// TIA Portal V17 export
// export: Created 2025-03-10T13:09:50.3447093Z, ExportSetting WithDefaults, DisplayName Totally Integrated Automation Portal, DisplayVersion V17 Update 8, DisplayName TIA Portal Openness, DisplayVersion V17 Update 8, DisplayName TIA Portal Version Control Interface, DisplayVersion V17, DisplayName SINAMICS Startdrive Advanced, DisplayVersion V17 SP2, DisplayName SINAMICS Startdrive G110M, G120, G120C, G120D, G120P, G115D, DisplayVersion V17 SP2, DisplayName SINAMICS Startdrive G130, G150, S120, S150, SINAMICS MV, S210, DisplayVersion V17 SP2, DisplayName STEP 7 Professional, DisplayVersion V17 Update 8, DisplayName SINUMERIK ONE STEP 7 Toolbox, DisplayVersion V17 Update 12, DisplayName SINUMERIK 840D sl STEP 7 Toolbox, DisplayVersion V17 Update 12, DisplayName STEP 7 Safety, DisplayVersion V17 Update 6, DisplayName WinCC Advanced, DisplayVersion V17 Update 8
FUNCTION "FC8004_UNIT_03_CLADDING" : Void   // FC8004, LAD
{ S7_Optimized_Access := 'FALSE' }
AUTHOR : ETXETAR
VERSION : 1.0
// stored: AutoNumber false, IsIECCheckEnabled false, SetENOAutomatically false, UDAEnableTagReadback false
   VAR_TEMP
      ZERO : Byte;   // ZERO
      STATUS_BLKMOV : Int;   // STATUS BLKMOV
      STATUS_FILL : Int;   // STATUS FILL
   END_VAR
   VAR CONSTANT
      FC_NUMBER : DInt := 8004;   // FC NUMBER
   END_VAR
   VAR_TEMP   // added for the SCL form of the ladder/FBD networks
      _w1 : Bool;
      _w2 : Bool;
      _w3 : Bool;
      _w4 : Bool;
   END_VAR
BEGIN

REGION Network 1: ZERO
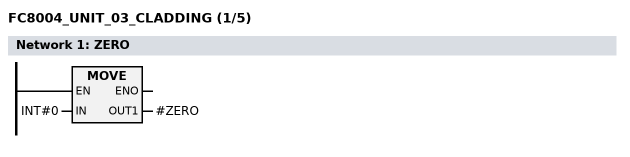
   RUNG wire#powerrail
      { S7_GenerateENO := "TRUE" } Move(in := INT#0, out1 => #ZERO)
   END_RUNG
   // the same network as SCL:
   #ZERO := INT#0;
END_REGION

REGION Network 2: HMI MANUAL PART A FIXTURE 1 STATUS
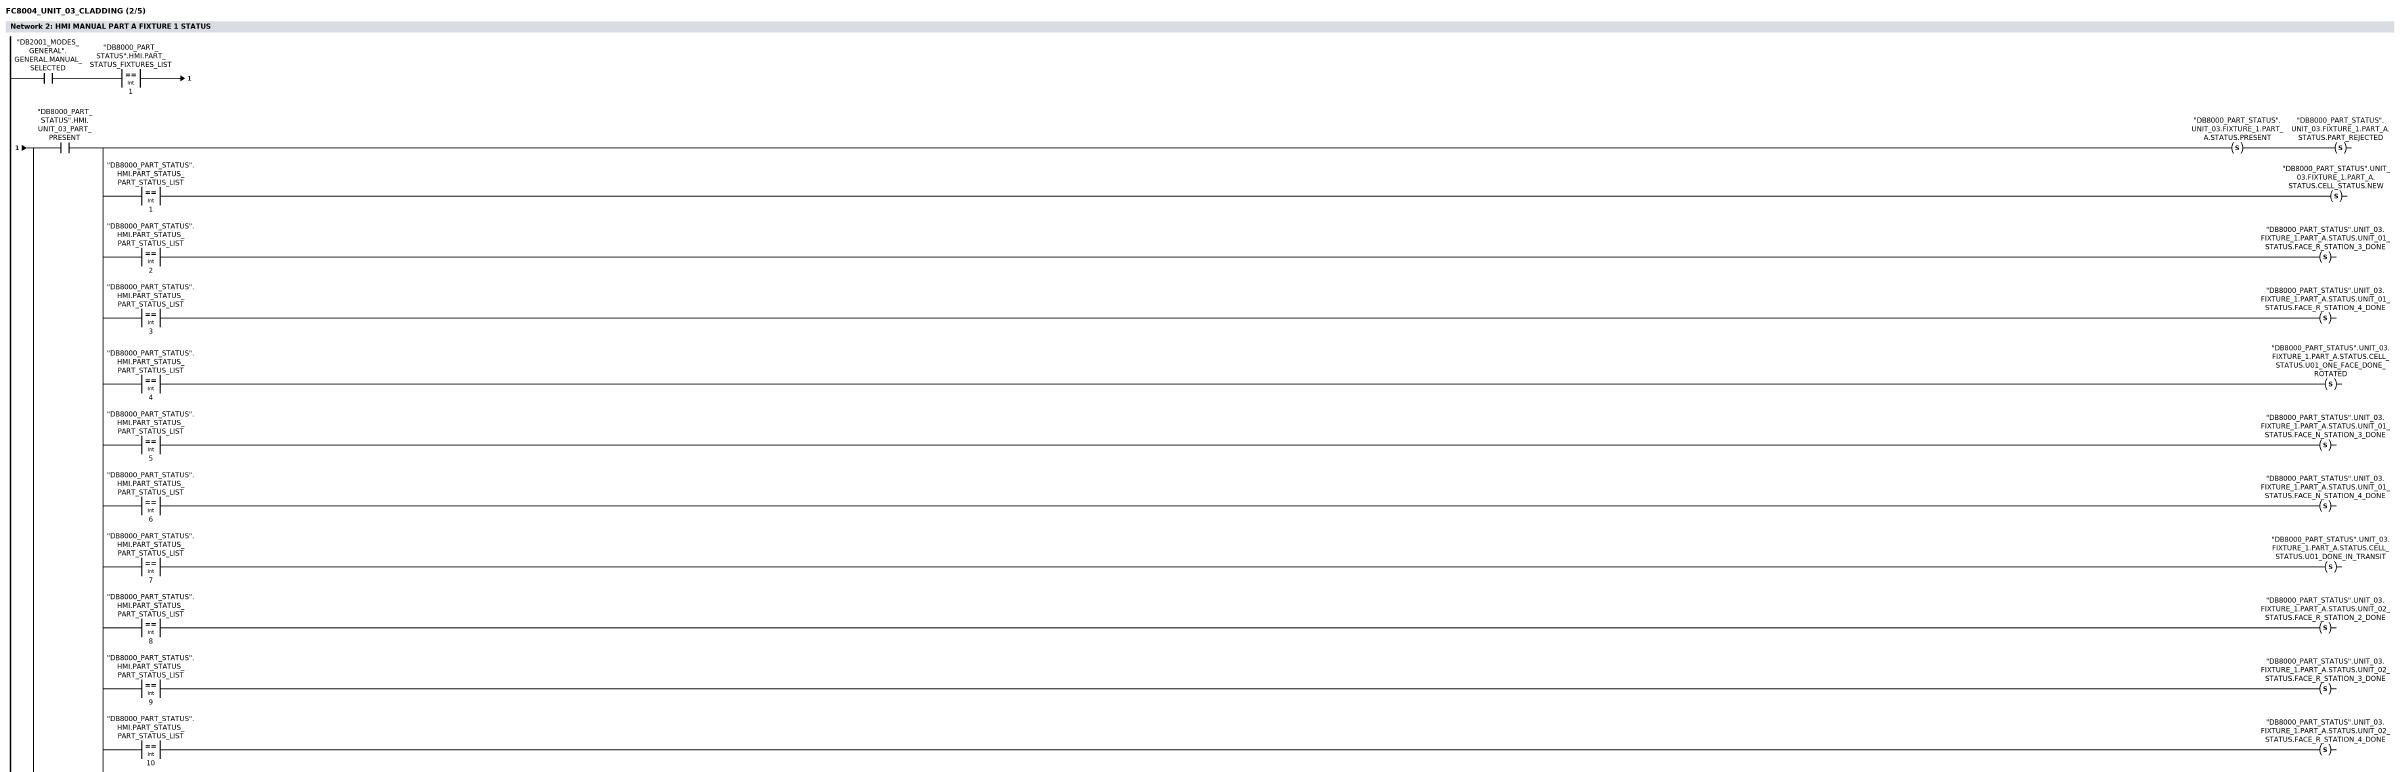
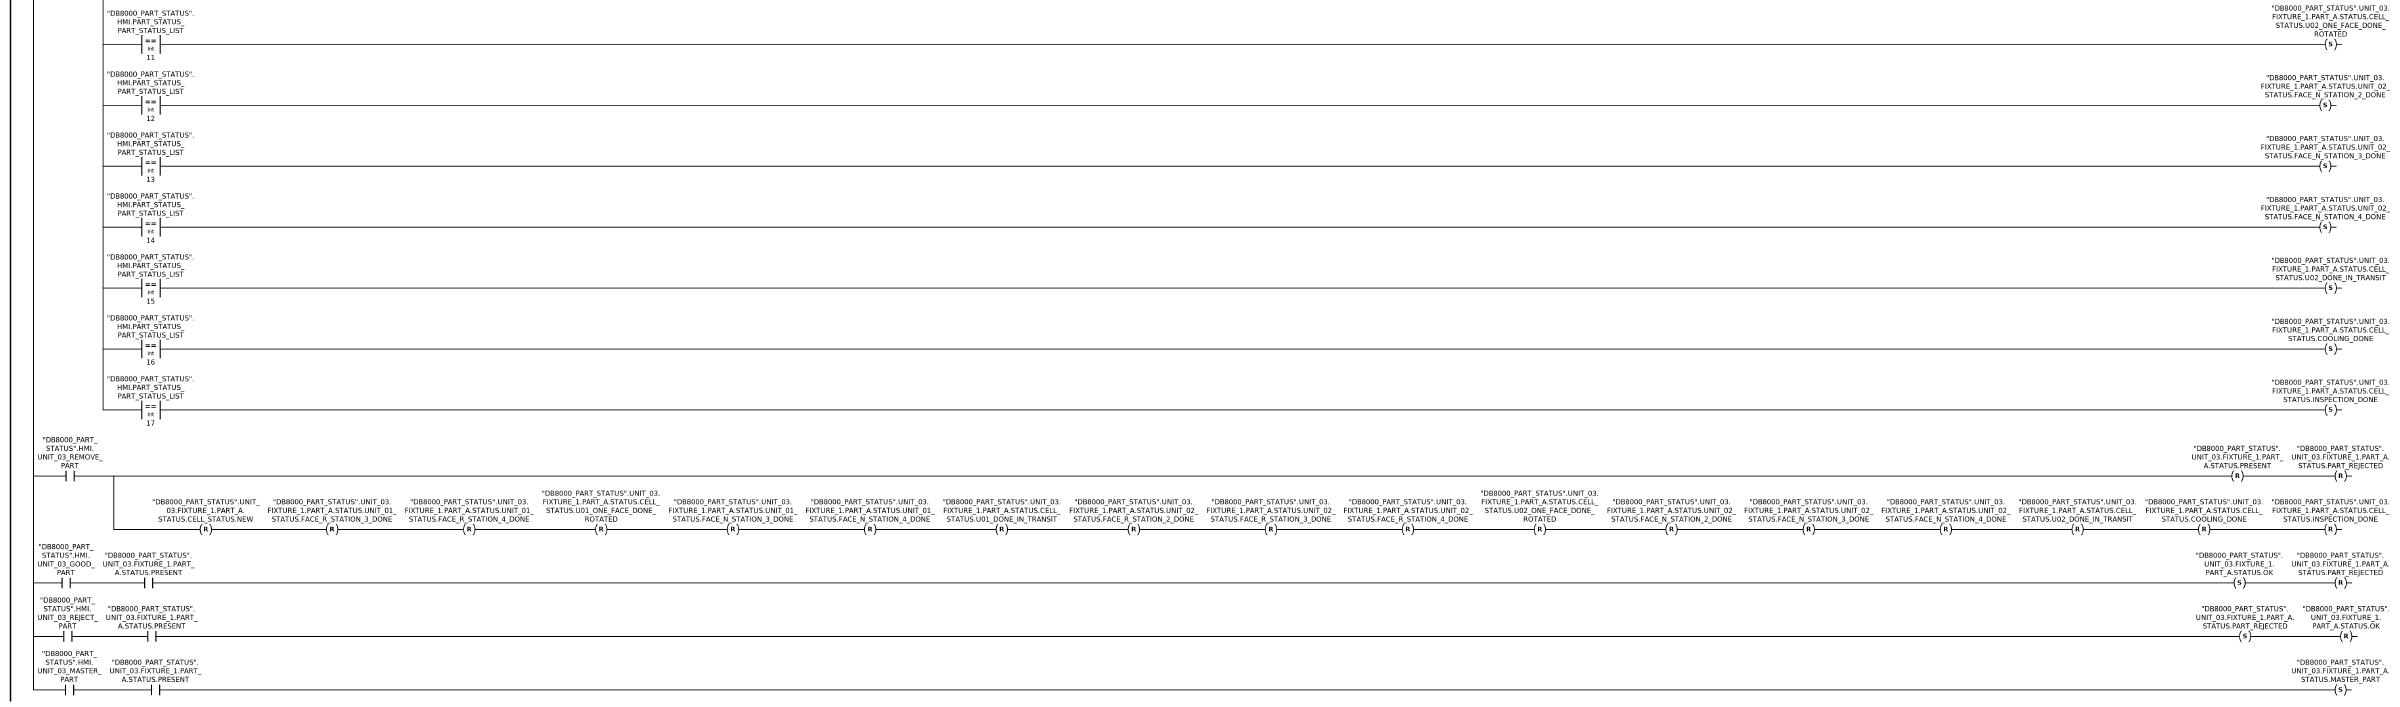
   RUNG wire#powerrail
      Contact( "DB2001_MODES_GENERAL".GENERAL.MANUAL_SELECTED )
      { S7_Templates := "SrcType := Int" } EQ_Contact(in1 := "DB8000_PART_STATUS".HMI.PART_STATUS_FIXTURES_LIST, in2 := 1)
      wire#w1
      Contact( "DB8000_PART_STATUS".HMI.UNIT_03_PART_PRESENT )
      wire#w2
      S_Coil( "DB8000_PART_STATUS".UNIT_03.FIXTURE_1.PART_A.STATUS.PRESENT )
      S_Coil( "DB8000_PART_STATUS".UNIT_03.FIXTURE_1.PART_A.STATUS.PART_REJECTED )
   END_RUNG
   RUNG wire#w2
      { S7_Templates := "SrcType := Int" } EQ_Contact(in1 := "DB8000_PART_STATUS".HMI.PART_STATUS_PART_STATUS_LIST, in2 := 1)
      S_Coil( "DB8000_PART_STATUS".UNIT_03.FIXTURE_1.PART_A.STATUS.CELL_STATUS.NEW )
   END_RUNG
   RUNG wire#w2
      { S7_Templates := "SrcType := Int" } EQ_Contact(in1 := "DB8000_PART_STATUS".HMI.PART_STATUS_PART_STATUS_LIST, in2 := 2)
      S_Coil( "DB8000_PART_STATUS".UNIT_03.FIXTURE_1.PART_A.STATUS.UNIT_01_STATUS.FACE_R_STATION_3_DONE )
   END_RUNG
   RUNG wire#w2
      { S7_Templates := "SrcType := Int" } EQ_Contact(in1 := "DB8000_PART_STATUS".HMI.PART_STATUS_PART_STATUS_LIST, in2 := 3)
      S_Coil( "DB8000_PART_STATUS".UNIT_03.FIXTURE_1.PART_A.STATUS.UNIT_01_STATUS.FACE_R_STATION_4_DONE )
   END_RUNG
   RUNG wire#w2
      { S7_Templates := "SrcType := Int" } EQ_Contact(in1 := "DB8000_PART_STATUS".HMI.PART_STATUS_PART_STATUS_LIST, in2 := 4)
      S_Coil( "DB8000_PART_STATUS".UNIT_03.FIXTURE_1.PART_A.STATUS.CELL_STATUS.U01_ONE_FACE_DONE_ROTATED )
   END_RUNG
   RUNG wire#w2
      { S7_Templates := "SrcType := Int" } EQ_Contact(in1 := "DB8000_PART_STATUS".HMI.PART_STATUS_PART_STATUS_LIST, in2 := 5)
      S_Coil( "DB8000_PART_STATUS".UNIT_03.FIXTURE_1.PART_A.STATUS.UNIT_01_STATUS.FACE_N_STATION_3_DONE )
   END_RUNG
   RUNG wire#w2
      { S7_Templates := "SrcType := Int" } EQ_Contact(in1 := "DB8000_PART_STATUS".HMI.PART_STATUS_PART_STATUS_LIST, in2 := 6)
      S_Coil( "DB8000_PART_STATUS".UNIT_03.FIXTURE_1.PART_A.STATUS.UNIT_01_STATUS.FACE_N_STATION_4_DONE )
   END_RUNG
   RUNG wire#w2
      { S7_Templates := "SrcType := Int" } EQ_Contact(in1 := "DB8000_PART_STATUS".HMI.PART_STATUS_PART_STATUS_LIST, in2 := 7)
      S_Coil( "DB8000_PART_STATUS".UNIT_03.FIXTURE_1.PART_A.STATUS.CELL_STATUS.U01_DONE_IN_TRANSIT )
   END_RUNG
   RUNG wire#w2
      { S7_Templates := "SrcType := Int" } EQ_Contact(in1 := "DB8000_PART_STATUS".HMI.PART_STATUS_PART_STATUS_LIST, in2 := 8)
      S_Coil( "DB8000_PART_STATUS".UNIT_03.FIXTURE_1.PART_A.STATUS.UNIT_02_STATUS.FACE_R_STATION_2_DONE )
   END_RUNG
   RUNG wire#w2
      { S7_Templates := "SrcType := Int" } EQ_Contact(in1 := "DB8000_PART_STATUS".HMI.PART_STATUS_PART_STATUS_LIST, in2 := 9)
      S_Coil( "DB8000_PART_STATUS".UNIT_03.FIXTURE_1.PART_A.STATUS.UNIT_02_STATUS.FACE_R_STATION_3_DONE )
   END_RUNG
   RUNG wire#w2
      { S7_Templates := "SrcType := Int" } EQ_Contact(in1 := "DB8000_PART_STATUS".HMI.PART_STATUS_PART_STATUS_LIST, in2 := 10)
      S_Coil( "DB8000_PART_STATUS".UNIT_03.FIXTURE_1.PART_A.STATUS.UNIT_02_STATUS.FACE_R_STATION_4_DONE )
   END_RUNG
   RUNG wire#w2
      { S7_Templates := "SrcType := Int" } EQ_Contact(in1 := "DB8000_PART_STATUS".HMI.PART_STATUS_PART_STATUS_LIST, in2 := 11)
      S_Coil( "DB8000_PART_STATUS".UNIT_03.FIXTURE_1.PART_A.STATUS.CELL_STATUS.U02_ONE_FACE_DONE_ROTATED )
   END_RUNG
   RUNG wire#w2
      { S7_Templates := "SrcType := Int" } EQ_Contact(in1 := "DB8000_PART_STATUS".HMI.PART_STATUS_PART_STATUS_LIST, in2 := 12)
      S_Coil( "DB8000_PART_STATUS".UNIT_03.FIXTURE_1.PART_A.STATUS.UNIT_02_STATUS.FACE_N_STATION_2_DONE )
   END_RUNG
   RUNG wire#w2
      { S7_Templates := "SrcType := Int" } EQ_Contact(in1 := "DB8000_PART_STATUS".HMI.PART_STATUS_PART_STATUS_LIST, in2 := 13)
      S_Coil( "DB8000_PART_STATUS".UNIT_03.FIXTURE_1.PART_A.STATUS.UNIT_02_STATUS.FACE_N_STATION_3_DONE )
   END_RUNG
   RUNG wire#w2
      { S7_Templates := "SrcType := Int" } EQ_Contact(in1 := "DB8000_PART_STATUS".HMI.PART_STATUS_PART_STATUS_LIST, in2 := 14)
      S_Coil( "DB8000_PART_STATUS".UNIT_03.FIXTURE_1.PART_A.STATUS.UNIT_02_STATUS.FACE_N_STATION_4_DONE )
   END_RUNG
   RUNG wire#w2
      { S7_Templates := "SrcType := Int" } EQ_Contact(in1 := "DB8000_PART_STATUS".HMI.PART_STATUS_PART_STATUS_LIST, in2 := 15)
      S_Coil( "DB8000_PART_STATUS".UNIT_03.FIXTURE_1.PART_A.STATUS.CELL_STATUS.U02_DONE_IN_TRANSIT )
   END_RUNG
   RUNG wire#w2
      { S7_Templates := "SrcType := Int" } EQ_Contact(in1 := "DB8000_PART_STATUS".HMI.PART_STATUS_PART_STATUS_LIST, in2 := 16)
      S_Coil( "DB8000_PART_STATUS".UNIT_03.FIXTURE_1.PART_A.STATUS.CELL_STATUS.COOLING_DONE )
   END_RUNG
   RUNG wire#w2
      { S7_Templates := "SrcType := Int" } EQ_Contact(in1 := "DB8000_PART_STATUS".HMI.PART_STATUS_PART_STATUS_LIST, in2 := 17)
      S_Coil( "DB8000_PART_STATUS".UNIT_03.FIXTURE_1.PART_A.STATUS.CELL_STATUS.INSPECTION_DONE )
   END_RUNG
   RUNG wire#w1
      Contact( "DB8000_PART_STATUS".HMI.UNIT_03_REMOVE_PART )
      wire#w3
      R_Coil( "DB8000_PART_STATUS".UNIT_03.FIXTURE_1.PART_A.STATUS.PRESENT )
      R_Coil( "DB8000_PART_STATUS".UNIT_03.FIXTURE_1.PART_A.STATUS.PART_REJECTED )
   END_RUNG
   RUNG wire#w3
      R_Coil( "DB8000_PART_STATUS".UNIT_03.FIXTURE_1.PART_A.STATUS.CELL_STATUS.NEW )
      R_Coil( "DB8000_PART_STATUS".UNIT_03.FIXTURE_1.PART_A.STATUS.UNIT_01_STATUS.FACE_R_STATION_3_DONE )
      R_Coil( "DB8000_PART_STATUS".UNIT_03.FIXTURE_1.PART_A.STATUS.UNIT_01_STATUS.FACE_R_STATION_4_DONE )
      R_Coil( "DB8000_PART_STATUS".UNIT_03.FIXTURE_1.PART_A.STATUS.CELL_STATUS.U01_ONE_FACE_DONE_ROTATED )
      R_Coil( "DB8000_PART_STATUS".UNIT_03.FIXTURE_1.PART_A.STATUS.UNIT_01_STATUS.FACE_N_STATION_3_DONE )
      R_Coil( "DB8000_PART_STATUS".UNIT_03.FIXTURE_1.PART_A.STATUS.UNIT_01_STATUS.FACE_N_STATION_4_DONE )
      R_Coil( "DB8000_PART_STATUS".UNIT_03.FIXTURE_1.PART_A.STATUS.CELL_STATUS.U01_DONE_IN_TRANSIT )
      R_Coil( "DB8000_PART_STATUS".UNIT_03.FIXTURE_1.PART_A.STATUS.UNIT_02_STATUS.FACE_R_STATION_2_DONE )
      R_Coil( "DB8000_PART_STATUS".UNIT_03.FIXTURE_1.PART_A.STATUS.UNIT_02_STATUS.FACE_R_STATION_3_DONE )
      R_Coil( "DB8000_PART_STATUS".UNIT_03.FIXTURE_1.PART_A.STATUS.UNIT_02_STATUS.FACE_R_STATION_4_DONE )
      R_Coil( "DB8000_PART_STATUS".UNIT_03.FIXTURE_1.PART_A.STATUS.CELL_STATUS.U02_ONE_FACE_DONE_ROTATED )
      R_Coil( "DB8000_PART_STATUS".UNIT_03.FIXTURE_1.PART_A.STATUS.UNIT_02_STATUS.FACE_N_STATION_2_DONE )
      R_Coil( "DB8000_PART_STATUS".UNIT_03.FIXTURE_1.PART_A.STATUS.UNIT_02_STATUS.FACE_N_STATION_3_DONE )
      R_Coil( "DB8000_PART_STATUS".UNIT_03.FIXTURE_1.PART_A.STATUS.UNIT_02_STATUS.FACE_N_STATION_4_DONE )
      R_Coil( "DB8000_PART_STATUS".UNIT_03.FIXTURE_1.PART_A.STATUS.CELL_STATUS.U02_DONE_IN_TRANSIT )
      R_Coil( "DB8000_PART_STATUS".UNIT_03.FIXTURE_1.PART_A.STATUS.CELL_STATUS.COOLING_DONE )
      R_Coil( "DB8000_PART_STATUS".UNIT_03.FIXTURE_1.PART_A.STATUS.CELL_STATUS.INSPECTION_DONE )
   END_RUNG
   RUNG wire#w1
      Contact( "DB8000_PART_STATUS".HMI.UNIT_03_GOOD_PART )
      Contact( "DB8000_PART_STATUS".UNIT_03.FIXTURE_1.PART_A.STATUS.PRESENT )
      S_Coil( "DB8000_PART_STATUS".UNIT_03.FIXTURE_1.PART_A.STATUS.OK )
      R_Coil( "DB8000_PART_STATUS".UNIT_03.FIXTURE_1.PART_A.STATUS.PART_REJECTED )
   END_RUNG
   RUNG wire#w1
      Contact( "DB8000_PART_STATUS".HMI.UNIT_03_REJECT_PART )
      Contact( "DB8000_PART_STATUS".UNIT_03.FIXTURE_1.PART_A.STATUS.PRESENT )
      S_Coil( "DB8000_PART_STATUS".UNIT_03.FIXTURE_1.PART_A.STATUS.PART_REJECTED )
      R_Coil( "DB8000_PART_STATUS".UNIT_03.FIXTURE_1.PART_A.STATUS.OK )
   END_RUNG
   RUNG wire#w1
      Contact( "DB8000_PART_STATUS".HMI.UNIT_03_MASTER_PART )
      Contact( "DB8000_PART_STATUS".UNIT_03.FIXTURE_1.PART_A.STATUS.PRESENT )
      S_Coil( "DB8000_PART_STATUS".UNIT_03.FIXTURE_1.PART_A.STATUS.MASTER_PART )
   END_RUNG
   // the same network as SCL:
   #_w1 := "DB2001_MODES_GENERAL".GENERAL.MANUAL_SELECTED AND ("DB8000_PART_STATUS".HMI.PART_STATUS_FIXTURES_LIST = 1);
   #_w2 := #_w1 AND "DB8000_PART_STATUS".HMI.UNIT_03_PART_PRESENT;
   IF #_w2 THEN
       "DB8000_PART_STATUS".UNIT_03.FIXTURE_1.PART_A.STATUS.PRESENT := TRUE;
       "DB8000_PART_STATUS".UNIT_03.FIXTURE_1.PART_A.STATUS.PART_REJECTED := TRUE;
   END_IF;
   IF #_w2 AND ("DB8000_PART_STATUS".HMI.PART_STATUS_PART_STATUS_LIST = 1) THEN
       "DB8000_PART_STATUS".UNIT_03.FIXTURE_1.PART_A.STATUS.CELL_STATUS.NEW := TRUE;
   END_IF;
   IF #_w2 AND ("DB8000_PART_STATUS".HMI.PART_STATUS_PART_STATUS_LIST = 2) THEN
       "DB8000_PART_STATUS".UNIT_03.FIXTURE_1.PART_A.STATUS.UNIT_01_STATUS.FACE_R_STATION_3_DONE := TRUE;
   END_IF;
   IF #_w2 AND ("DB8000_PART_STATUS".HMI.PART_STATUS_PART_STATUS_LIST = 3) THEN
       "DB8000_PART_STATUS".UNIT_03.FIXTURE_1.PART_A.STATUS.UNIT_01_STATUS.FACE_R_STATION_4_DONE := TRUE;
   END_IF;
   IF #_w2 AND ("DB8000_PART_STATUS".HMI.PART_STATUS_PART_STATUS_LIST = 4) THEN
       "DB8000_PART_STATUS".UNIT_03.FIXTURE_1.PART_A.STATUS.CELL_STATUS.U01_ONE_FACE_DONE_ROTATED := TRUE;
   END_IF;
   IF #_w2 AND ("DB8000_PART_STATUS".HMI.PART_STATUS_PART_STATUS_LIST = 5) THEN
       "DB8000_PART_STATUS".UNIT_03.FIXTURE_1.PART_A.STATUS.UNIT_01_STATUS.FACE_N_STATION_3_DONE := TRUE;
   END_IF;
   IF #_w2 AND ("DB8000_PART_STATUS".HMI.PART_STATUS_PART_STATUS_LIST = 6) THEN
       "DB8000_PART_STATUS".UNIT_03.FIXTURE_1.PART_A.STATUS.UNIT_01_STATUS.FACE_N_STATION_4_DONE := TRUE;
   END_IF;
   IF #_w2 AND ("DB8000_PART_STATUS".HMI.PART_STATUS_PART_STATUS_LIST = 7) THEN
       "DB8000_PART_STATUS".UNIT_03.FIXTURE_1.PART_A.STATUS.CELL_STATUS.U01_DONE_IN_TRANSIT := TRUE;
   END_IF;
   IF #_w2 AND ("DB8000_PART_STATUS".HMI.PART_STATUS_PART_STATUS_LIST = 8) THEN
       "DB8000_PART_STATUS".UNIT_03.FIXTURE_1.PART_A.STATUS.UNIT_02_STATUS.FACE_R_STATION_2_DONE := TRUE;
   END_IF;
   IF #_w2 AND ("DB8000_PART_STATUS".HMI.PART_STATUS_PART_STATUS_LIST = 9) THEN
       "DB8000_PART_STATUS".UNIT_03.FIXTURE_1.PART_A.STATUS.UNIT_02_STATUS.FACE_R_STATION_3_DONE := TRUE;
   END_IF;
   IF #_w2 AND ("DB8000_PART_STATUS".HMI.PART_STATUS_PART_STATUS_LIST = 10) THEN
       "DB8000_PART_STATUS".UNIT_03.FIXTURE_1.PART_A.STATUS.UNIT_02_STATUS.FACE_R_STATION_4_DONE := TRUE;
   END_IF;
   IF #_w2 AND ("DB8000_PART_STATUS".HMI.PART_STATUS_PART_STATUS_LIST = 11) THEN
       "DB8000_PART_STATUS".UNIT_03.FIXTURE_1.PART_A.STATUS.CELL_STATUS.U02_ONE_FACE_DONE_ROTATED := TRUE;
   END_IF;
   IF #_w2 AND ("DB8000_PART_STATUS".HMI.PART_STATUS_PART_STATUS_LIST = 12) THEN
       "DB8000_PART_STATUS".UNIT_03.FIXTURE_1.PART_A.STATUS.UNIT_02_STATUS.FACE_N_STATION_2_DONE := TRUE;
   END_IF;
   IF #_w2 AND ("DB8000_PART_STATUS".HMI.PART_STATUS_PART_STATUS_LIST = 13) THEN
       "DB8000_PART_STATUS".UNIT_03.FIXTURE_1.PART_A.STATUS.UNIT_02_STATUS.FACE_N_STATION_3_DONE := TRUE;
   END_IF;
   IF #_w2 AND ("DB8000_PART_STATUS".HMI.PART_STATUS_PART_STATUS_LIST = 14) THEN
       "DB8000_PART_STATUS".UNIT_03.FIXTURE_1.PART_A.STATUS.UNIT_02_STATUS.FACE_N_STATION_4_DONE := TRUE;
   END_IF;
   IF #_w2 AND ("DB8000_PART_STATUS".HMI.PART_STATUS_PART_STATUS_LIST = 15) THEN
       "DB8000_PART_STATUS".UNIT_03.FIXTURE_1.PART_A.STATUS.CELL_STATUS.U02_DONE_IN_TRANSIT := TRUE;
   END_IF;
   IF #_w2 AND ("DB8000_PART_STATUS".HMI.PART_STATUS_PART_STATUS_LIST = 16) THEN
       "DB8000_PART_STATUS".UNIT_03.FIXTURE_1.PART_A.STATUS.CELL_STATUS.COOLING_DONE := TRUE;
   END_IF;
   IF #_w2 AND ("DB8000_PART_STATUS".HMI.PART_STATUS_PART_STATUS_LIST = 17) THEN
       "DB8000_PART_STATUS".UNIT_03.FIXTURE_1.PART_A.STATUS.CELL_STATUS.INSPECTION_DONE := TRUE;
   END_IF;
   IF #_w1 AND "DB8000_PART_STATUS".HMI.UNIT_03_REMOVE_PART THEN
       "DB8000_PART_STATUS".UNIT_03.FIXTURE_1.PART_A.STATUS.PRESENT := FALSE;
       "DB8000_PART_STATUS".UNIT_03.FIXTURE_1.PART_A.STATUS.PART_REJECTED := FALSE;
       "DB8000_PART_STATUS".UNIT_03.FIXTURE_1.PART_A.STATUS.CELL_STATUS.NEW := FALSE;
       "DB8000_PART_STATUS".UNIT_03.FIXTURE_1.PART_A.STATUS.UNIT_01_STATUS.FACE_R_STATION_3_DONE := FALSE;
       "DB8000_PART_STATUS".UNIT_03.FIXTURE_1.PART_A.STATUS.UNIT_01_STATUS.FACE_R_STATION_4_DONE := FALSE;
       "DB8000_PART_STATUS".UNIT_03.FIXTURE_1.PART_A.STATUS.CELL_STATUS.U01_ONE_FACE_DONE_ROTATED := FALSE;
       "DB8000_PART_STATUS".UNIT_03.FIXTURE_1.PART_A.STATUS.UNIT_01_STATUS.FACE_N_STATION_3_DONE := FALSE;
       "DB8000_PART_STATUS".UNIT_03.FIXTURE_1.PART_A.STATUS.UNIT_01_STATUS.FACE_N_STATION_4_DONE := FALSE;
       "DB8000_PART_STATUS".UNIT_03.FIXTURE_1.PART_A.STATUS.CELL_STATUS.U01_DONE_IN_TRANSIT := FALSE;
       "DB8000_PART_STATUS".UNIT_03.FIXTURE_1.PART_A.STATUS.UNIT_02_STATUS.FACE_R_STATION_2_DONE := FALSE;
       "DB8000_PART_STATUS".UNIT_03.FIXTURE_1.PART_A.STATUS.UNIT_02_STATUS.FACE_R_STATION_3_DONE := FALSE;
       "DB8000_PART_STATUS".UNIT_03.FIXTURE_1.PART_A.STATUS.UNIT_02_STATUS.FACE_R_STATION_4_DONE := FALSE;
       "DB8000_PART_STATUS".UNIT_03.FIXTURE_1.PART_A.STATUS.CELL_STATUS.U02_ONE_FACE_DONE_ROTATED := FALSE;
       "DB8000_PART_STATUS".UNIT_03.FIXTURE_1.PART_A.STATUS.UNIT_02_STATUS.FACE_N_STATION_2_DONE := FALSE;
       "DB8000_PART_STATUS".UNIT_03.FIXTURE_1.PART_A.STATUS.UNIT_02_STATUS.FACE_N_STATION_3_DONE := FALSE;
       "DB8000_PART_STATUS".UNIT_03.FIXTURE_1.PART_A.STATUS.UNIT_02_STATUS.FACE_N_STATION_4_DONE := FALSE;
       "DB8000_PART_STATUS".UNIT_03.FIXTURE_1.PART_A.STATUS.CELL_STATUS.U02_DONE_IN_TRANSIT := FALSE;
       "DB8000_PART_STATUS".UNIT_03.FIXTURE_1.PART_A.STATUS.CELL_STATUS.COOLING_DONE := FALSE;
       "DB8000_PART_STATUS".UNIT_03.FIXTURE_1.PART_A.STATUS.CELL_STATUS.INSPECTION_DONE := FALSE;
   END_IF;
   IF #_w1 AND "DB8000_PART_STATUS".HMI.UNIT_03_GOOD_PART AND "DB8000_PART_STATUS".UNIT_03.FIXTURE_1.PART_A.STATUS.PRESENT THEN
       "DB8000_PART_STATUS".UNIT_03.FIXTURE_1.PART_A.STATUS.OK := TRUE;
       "DB8000_PART_STATUS".UNIT_03.FIXTURE_1.PART_A.STATUS.PART_REJECTED := FALSE;
   END_IF;
   IF #_w1 AND "DB8000_PART_STATUS".HMI.UNIT_03_REJECT_PART AND "DB8000_PART_STATUS".UNIT_03.FIXTURE_1.PART_A.STATUS.PRESENT THEN
       "DB8000_PART_STATUS".UNIT_03.FIXTURE_1.PART_A.STATUS.PART_REJECTED := TRUE;
       "DB8000_PART_STATUS".UNIT_03.FIXTURE_1.PART_A.STATUS.OK := FALSE;
   END_IF;
   IF #_w1 AND "DB8000_PART_STATUS".HMI.UNIT_03_MASTER_PART AND "DB8000_PART_STATUS".UNIT_03.FIXTURE_1.PART_A.STATUS.PRESENT THEN
       "DB8000_PART_STATUS".UNIT_03.FIXTURE_1.PART_A.STATUS.MASTER_PART := TRUE;
   END_IF;
END_REGION

REGION Network 3: OPERATOR HELP
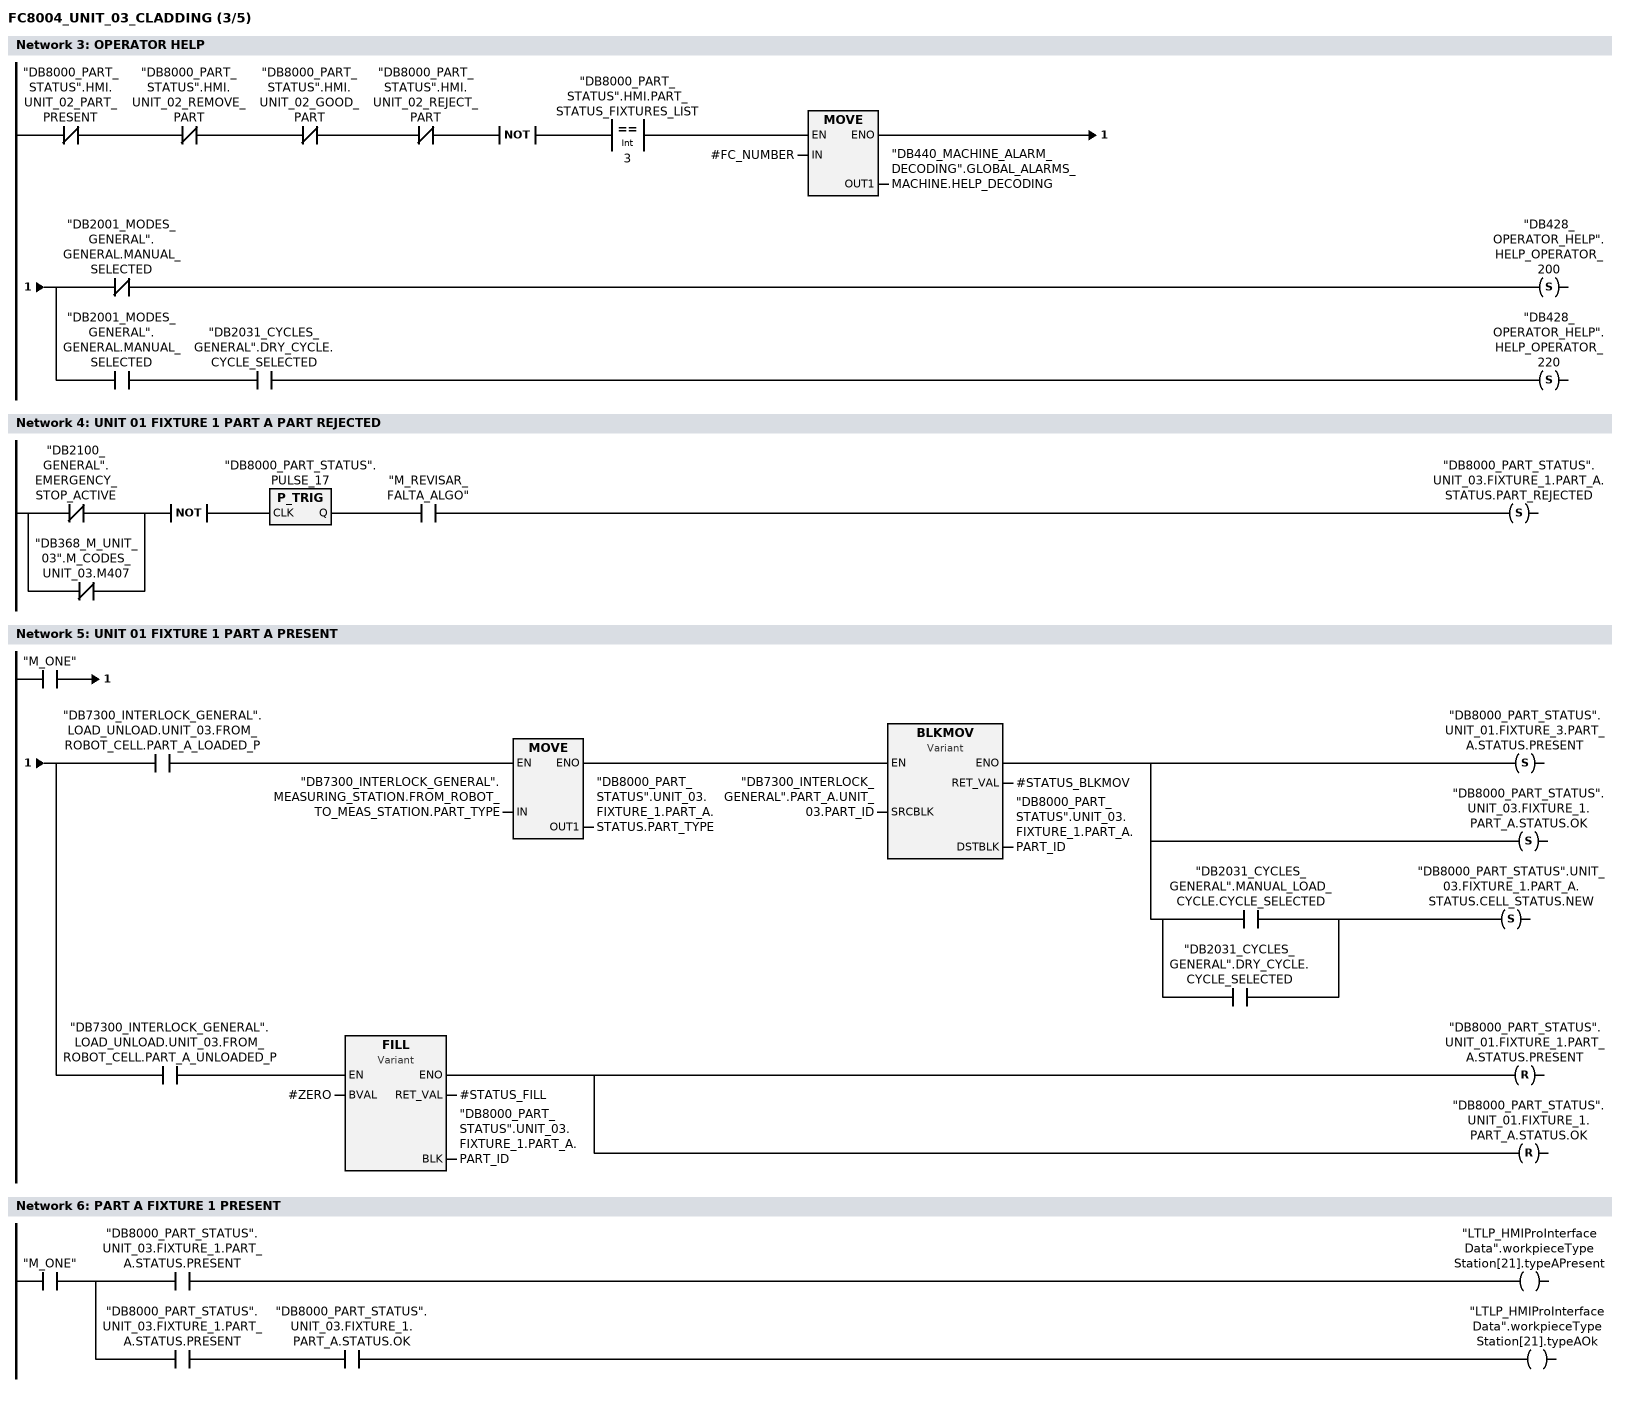
   RUNG wire#powerrail
      I_Contact( "DB8000_PART_STATUS".HMI.UNIT_02_PART_PRESENT )
      I_Contact( "DB8000_PART_STATUS".HMI.UNIT_02_REMOVE_PART )
      I_Contact( "DB8000_PART_STATUS".HMI.UNIT_02_GOOD_PART )
      I_Contact( "DB8000_PART_STATUS".HMI.UNIT_02_REJECT_PART )
      Not()
      { S7_Templates := "SrcType := Int" } EQ_Contact(in1 := "DB8000_PART_STATUS".HMI.PART_STATUS_FIXTURES_LIST, in2 := 3)
      { S7_GenerateENO := "TRUE" } Move(in := #FC_NUMBER, out1 => "DB440_MACHINE_ALARM_DECODING".GLOBAL_ALARMS_MACHINE.HELP_DECODING)
      wire#w1
      I_Contact( "DB2001_MODES_GENERAL".GENERAL.MANUAL_SELECTED )
      S_Coil( "DB428_OPERATOR_HELP".HELP_OPERATOR_200 )
   END_RUNG
   RUNG wire#w1
      Contact( "DB2001_MODES_GENERAL".GENERAL.MANUAL_SELECTED )
      Contact( "DB2031_CYCLES_GENERAL".DRY_CYCLE.CYCLE_SELECTED )
      S_Coil( "DB428_OPERATOR_HELP".HELP_OPERATOR_220 )
   END_RUNG
   // the same network as SCL:
   // ENO of a box is taken as its EN; it also drops when the box reports an error
   #_w1 := NOT (NOT "DB8000_PART_STATUS".HMI.UNIT_02_PART_PRESENT AND NOT "DB8000_PART_STATUS".HMI.UNIT_02_REMOVE_PART AND NOT "DB8000_PART_STATUS".HMI.UNIT_02_GOOD_PART AND NOT "DB8000_PART_STATUS".HMI.UNIT_02_REJECT_PART) AND ("DB8000_PART_STATUS".HMI.PART_STATUS_FIXTURES_LIST = 3);
   IF #_w1 THEN "DB440_MACHINE_ALARM_DECODING".GLOBAL_ALARMS_MACHINE.HELP_DECODING := #FC_NUMBER; END_IF;
   IF #_w1 AND NOT "DB2001_MODES_GENERAL".GENERAL.MANUAL_SELECTED THEN
       "DB428_OPERATOR_HELP".HELP_OPERATOR_200 := TRUE;
   END_IF;
   IF #_w1 AND "DB2001_MODES_GENERAL".GENERAL.MANUAL_SELECTED AND "DB2031_CYCLES_GENERAL".DRY_CYCLE.CYCLE_SELECTED THEN
       "DB428_OPERATOR_HELP".HELP_OPERATOR_220 := TRUE;
   END_IF;
END_REGION

REGION Network 4: UNIT 01 FIXTURE 1 PART A PART REJECTED
   RUNG wire#powerrail
      I_Contact( "DB2100_GENERAL".EMERGENCY_STOP_ACTIVE )
      wire#w1
      Not()
      P_Trig( "DB8000_PART_STATUS".PULSE_17 )
      Contact( "M_REVISAR_FALTA_ALGO" )
      S_Coil( "DB8000_PART_STATUS".UNIT_03.FIXTURE_1.PART_A.STATUS.PART_REJECTED )
   END_RUNG
   RUNG wire#powerrail
      I_Contact( "DB368_M_UNIT_03".M_CODES_UNIT_03.M407 )
   END_RUNG wire#w1
   // the same network as SCL:
   #_w1 := NOT (NOT "DB2100_GENERAL".EMERGENCY_STOP_ACTIVE OR NOT "DB368_M_UNIT_03".M_CODES_UNIT_03.M407);
   #_w2 := #_w1 AND NOT "DB8000_PART_STATUS".PULSE_17;   // rising edge
   "DB8000_PART_STATUS".PULSE_17 := #_w1;
   IF #_w2 AND "M_REVISAR_FALTA_ALGO" THEN
       "DB8000_PART_STATUS".UNIT_03.FIXTURE_1.PART_A.STATUS.PART_REJECTED := TRUE;
   END_IF;
END_REGION

REGION Network 5: UNIT 01 FIXTURE 1 PART A PRESENT
   RUNG wire#powerrail
      Contact( "M_ONE" )
      wire#w1
      Contact( "DB7300_INTERLOCK_GENERAL".LOAD_UNLOAD.UNIT_03.FROM_ROBOT_CELL.PART_A_LOADED_P )
      { S7_GenerateENO := "TRUE" } Move(in := "DB7300_INTERLOCK_GENERAL".MEASURING_STATION.FROM_ROBOT_TO_MEAS_STATION.PART_TYPE, out1 => "DB8000_PART_STATUS".UNIT_03.FIXTURE_1.PART_A.STATUS.PART_TYPE)
      { S7_Templates := "blk_type := Variant" } BLKMOV(SRCBLK := "DB7300_INTERLOCK_GENERAL".PART_A.UNIT_03.PART_ID, RET_VAL => #STATUS_BLKMOV, DSTBLK => "DB8000_PART_STATUS".UNIT_03.FIXTURE_1.PART_A.PART_ID)
      wire#w2
      S_Coil( "DB8000_PART_STATUS".UNIT_01.FIXTURE_3.PART_A.STATUS.PRESENT )
   END_RUNG
   RUNG wire#w2
      S_Coil( "DB8000_PART_STATUS".UNIT_03.FIXTURE_1.PART_A.STATUS.OK )
   END_RUNG
   RUNG wire#w2
      Contact( "DB2031_CYCLES_GENERAL".MANUAL_LOAD_CYCLE.CYCLE_SELECTED )
      wire#w3
      S_Coil( "DB8000_PART_STATUS".UNIT_03.FIXTURE_1.PART_A.STATUS.CELL_STATUS.NEW )
   END_RUNG
   RUNG wire#w2
      Contact( "DB2031_CYCLES_GENERAL".DRY_CYCLE.CYCLE_SELECTED )
   END_RUNG wire#w3
   RUNG wire#w1
      Contact( "DB7300_INTERLOCK_GENERAL".LOAD_UNLOAD.UNIT_03.FROM_ROBOT_CELL.PART_A_UNLOADED_P )
      { S7_Templates := "ptr_type := Variant" } FILL(BVAL := #ZERO, RET_VAL => #STATUS_FILL, BLK => "DB8000_PART_STATUS".UNIT_03.FIXTURE_1.PART_A.PART_ID)
      wire#w4
      R_Coil( "DB8000_PART_STATUS".UNIT_01.FIXTURE_1.PART_A.STATUS.PRESENT )
   END_RUNG
   RUNG wire#w4
      R_Coil( "DB8000_PART_STATUS".UNIT_01.FIXTURE_1.PART_A.STATUS.OK )
   END_RUNG
   // the same network as SCL:
   // ENO of a box is taken as its EN; it also drops when the box reports an error
   #_w1 := "M_ONE" AND "DB7300_INTERLOCK_GENERAL".LOAD_UNLOAD.UNIT_03.FROM_ROBOT_CELL.PART_A_LOADED_P;
   IF #_w1 THEN
       "DB8000_PART_STATUS".UNIT_03.FIXTURE_1.PART_A.STATUS.PART_TYPE := "DB7300_INTERLOCK_GENERAL".MEASURING_STATION.FROM_ROBOT_TO_MEAS_STATION.PART_TYPE;
   END_IF;
   #_w3 := "M_ONE";
   #STATUS_BLKMOV := BLKMOV(EN := #_w1,
                           SRCBLK := "DB7300_INTERLOCK_GENERAL".PART_A.UNIT_03.PART_ID,
                           DSTBLK => "DB8000_PART_STATUS".UNIT_03.FIXTURE_1.PART_A.PART_ID,
                           ENO => #_w2);
   IF #_w2 THEN
       "DB8000_PART_STATUS".UNIT_01.FIXTURE_3.PART_A.STATUS.PRESENT := TRUE;
       "DB8000_PART_STATUS".UNIT_03.FIXTURE_1.PART_A.STATUS.OK := TRUE;
   END_IF;
   IF #_w2 AND ("DB2031_CYCLES_GENERAL".MANUAL_LOAD_CYCLE.CYCLE_SELECTED OR "DB2031_CYCLES_GENERAL".DRY_CYCLE.CYCLE_SELECTED) THEN
       "DB8000_PART_STATUS".UNIT_03.FIXTURE_1.PART_A.STATUS.CELL_STATUS.NEW := TRUE;
   END_IF;
   #STATUS_FILL := FILL(EN := #_w3 AND "DB7300_INTERLOCK_GENERAL".LOAD_UNLOAD.UNIT_03.FROM_ROBOT_CELL.PART_A_UNLOADED_P,
                        BVAL := #ZERO,
                        BLK => "DB8000_PART_STATUS".UNIT_03.FIXTURE_1.PART_A.PART_ID,
                        ENO => #_w4);
   IF #_w4 THEN
       "DB8000_PART_STATUS".UNIT_01.FIXTURE_1.PART_A.STATUS.PRESENT := FALSE;
       "DB8000_PART_STATUS".UNIT_01.FIXTURE_1.PART_A.STATUS.OK := FALSE;
   END_IF;
END_REGION

REGION Network 6: PART A FIXTURE 1 PRESENT
   RUNG wire#powerrail
      Contact( "M_ONE" )
      wire#w1
      Contact( "DB8000_PART_STATUS".UNIT_03.FIXTURE_1.PART_A.STATUS.PRESENT )
      Coil( "LTLP_HMIProInterfaceData".workpieceTypeStation[21].typeAPresent )
   END_RUNG
   RUNG wire#w1
      Contact( "DB8000_PART_STATUS".UNIT_03.FIXTURE_1.PART_A.STATUS.PRESENT )
      Contact( "DB8000_PART_STATUS".UNIT_03.FIXTURE_1.PART_A.STATUS.OK )
      Coil( "LTLP_HMIProInterfaceData".workpieceTypeStation[21].typeAOk )
   END_RUNG
   // the same network as SCL:
   "LTLP_HMIProInterfaceData".workpieceTypeStation[21].typeAPresent := "M_ONE" AND "DB8000_PART_STATUS".UNIT_03.FIXTURE_1.PART_A.STATUS.PRESENT;
   "LTLP_HMIProInterfaceData".workpieceTypeStation[21].typeAOk := "M_ONE" AND "DB8000_PART_STATUS".UNIT_03.FIXTURE_1.PART_A.STATUS.PRESENT AND "DB8000_PART_STATUS".UNIT_03.FIXTURE_1.PART_A.STATUS.OK;
END_REGION

REGION Network 7: PART A FIXTURE 1 RESET STATUS TO ZERO
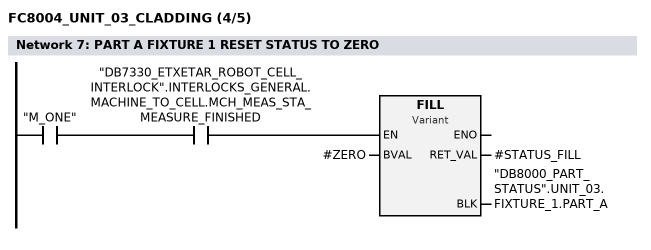
   RUNG wire#powerrail
      Contact( "M_ONE" )
      Contact( "DB7330_ETXETAR_ROBOT_CELL_INTERLOCK".INTERLOCKS_GENERAL.MACHINE_TO_CELL.MCH_MEAS_STA_MEASURE_FINISHED )
      { S7_Templates := "ptr_type := Variant" } FILL(BVAL := #ZERO, RET_VAL => #STATUS_FILL, BLK => "DB8000_PART_STATUS".UNIT_03.FIXTURE_1.PART_A)
   END_RUNG
   // the same network as SCL:
   IF "M_ONE" AND "DB7330_ETXETAR_ROBOT_CELL_INTERLOCK".INTERLOCKS_GENERAL.MACHINE_TO_CELL.MCH_MEAS_STA_MEASURE_FINISHED THEN
       #STATUS_FILL := FILL(BVAL := #ZERO, BLK => "DB8000_PART_STATUS".UNIT_03.FIXTURE_1.PART_A);
   END_IF;
END_REGION

REGION Network 8: PART A FIXTURE 1 COLOR STATUS
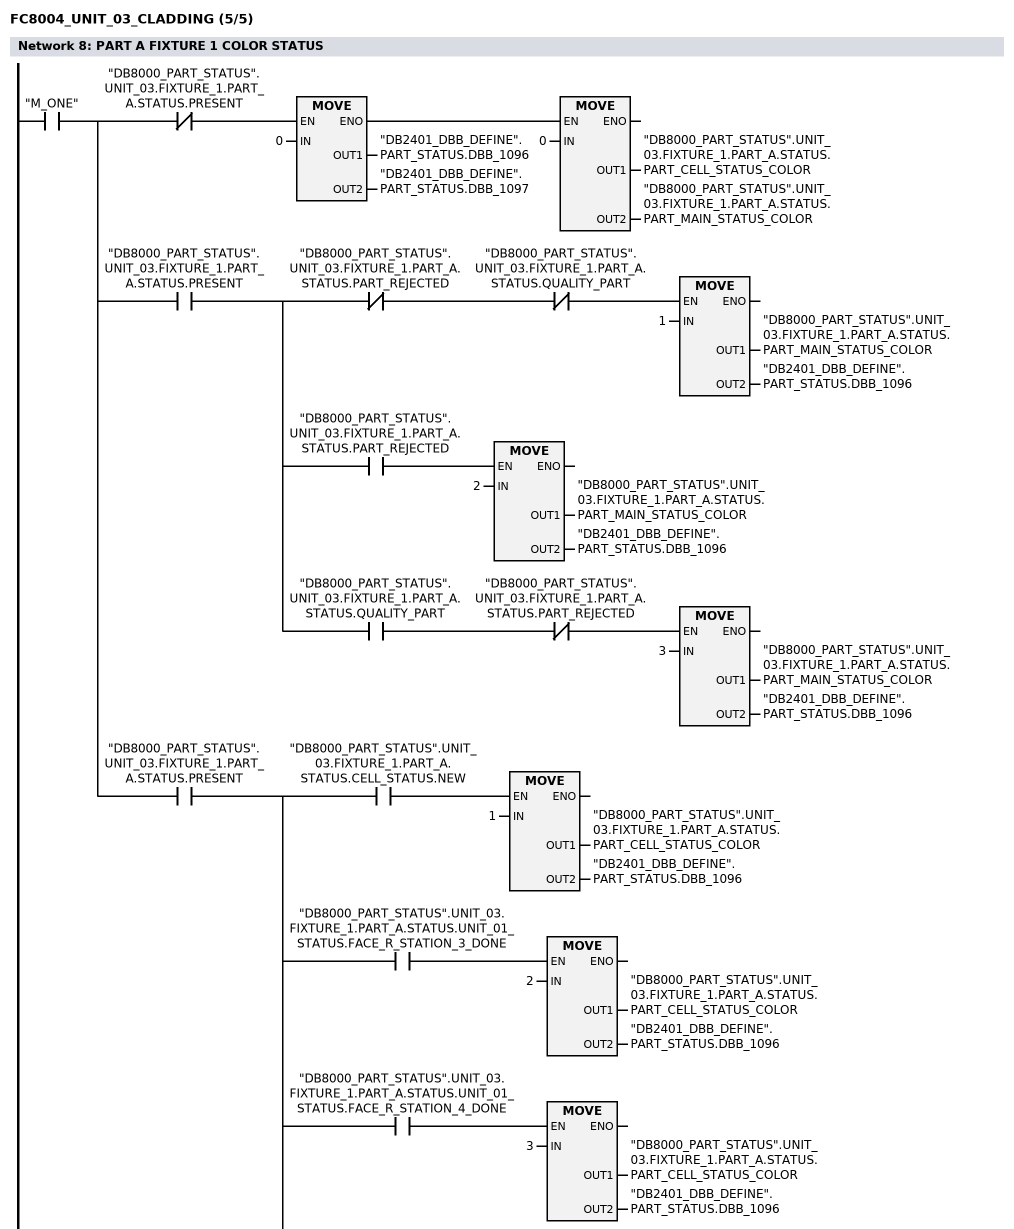
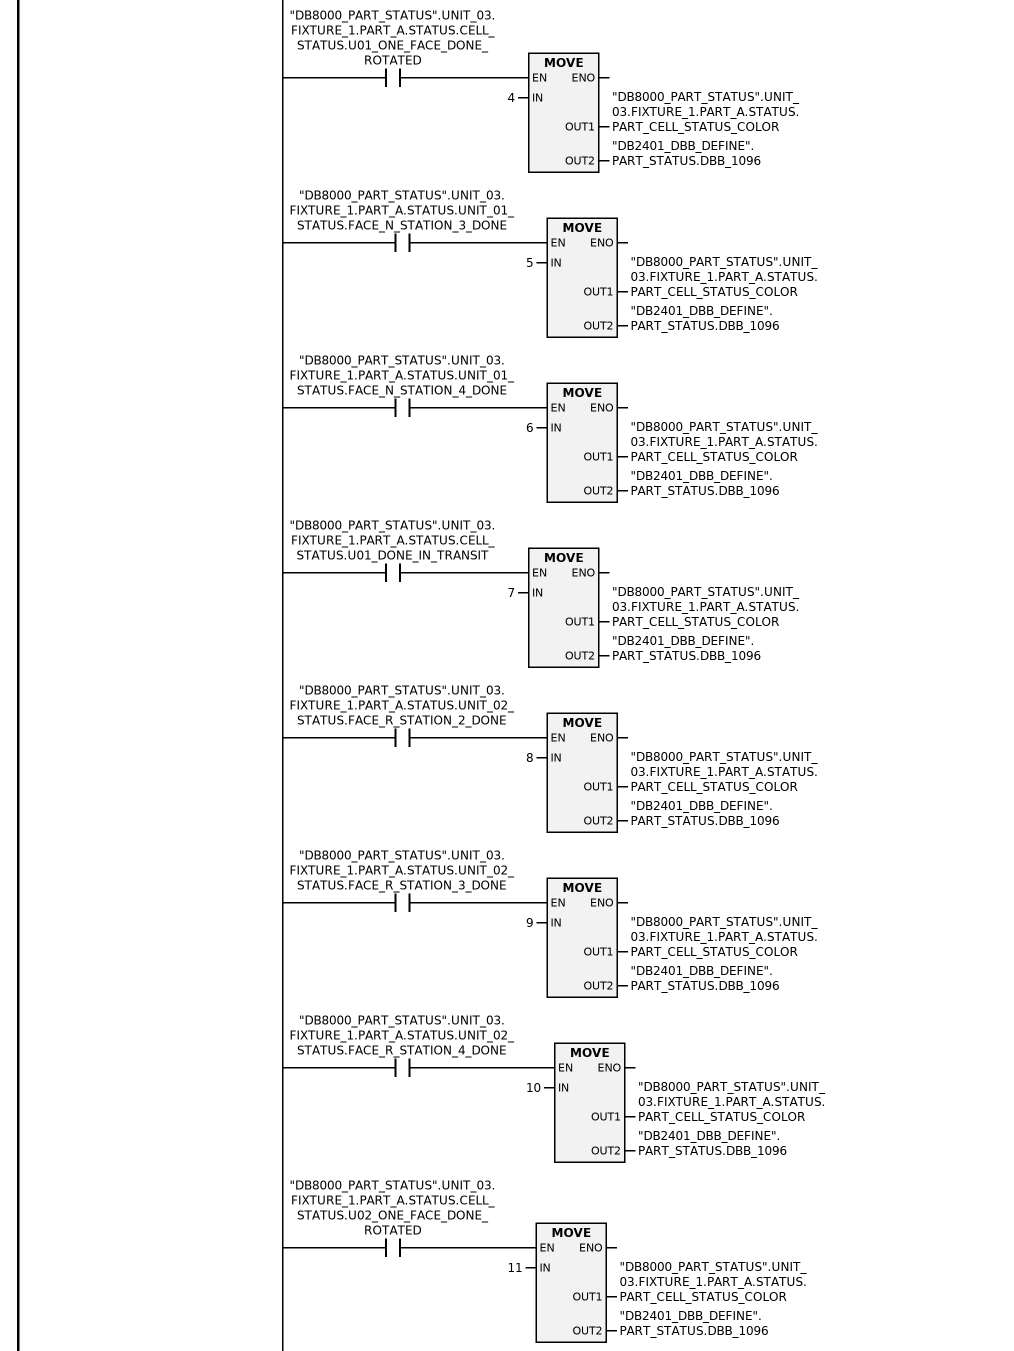
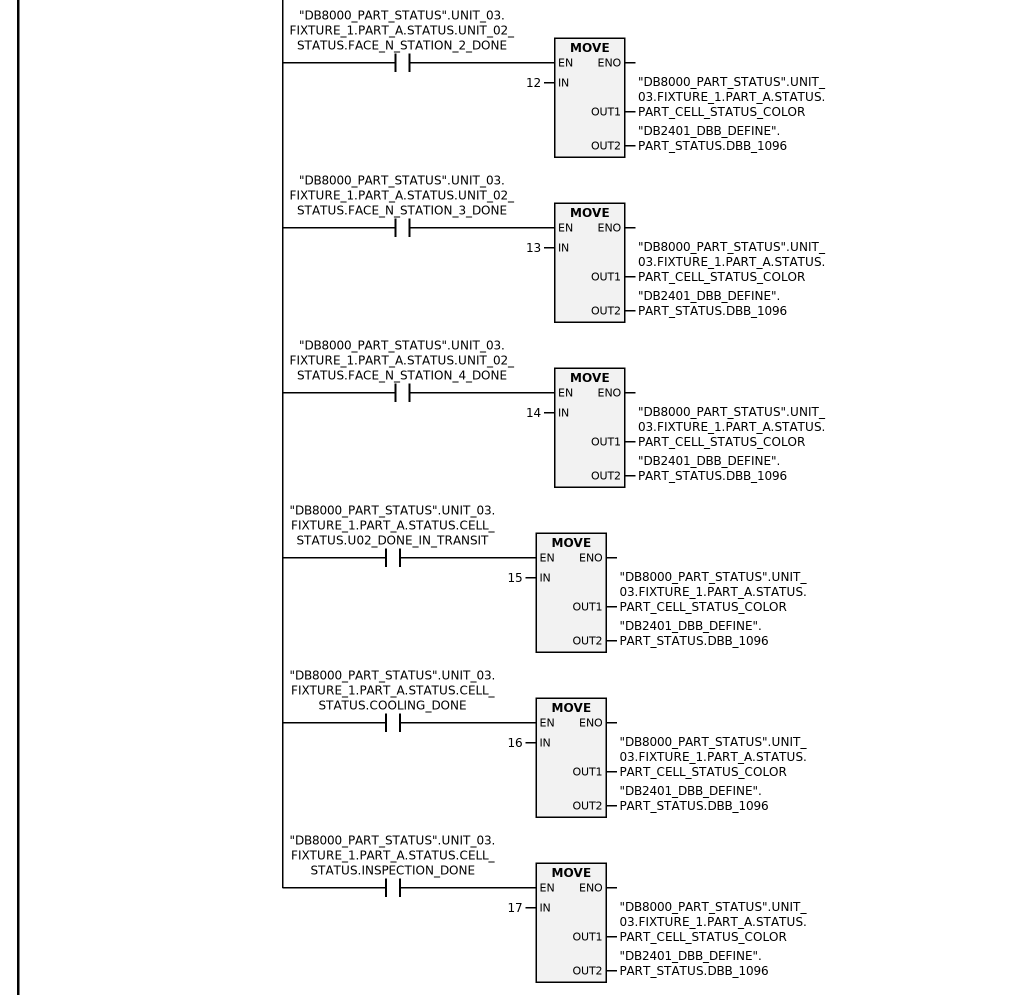
   RUNG wire#powerrail
      Contact( "M_ONE" )
      wire#w1
      I_Contact( "DB8000_PART_STATUS".UNIT_03.FIXTURE_1.PART_A.STATUS.PRESENT )
      { S7_GenerateENO := "TRUE" } Move(in := 0, out1 => "DB2401_DBB_DEFINE".PART_STATUS.DBB_1096, out2 => "DB2401_DBB_DEFINE".PART_STATUS.DBB_1097)
      { S7_GenerateENO := "TRUE" } Move(in := 0, out1 => "DB8000_PART_STATUS".UNIT_03.FIXTURE_1.PART_A.STATUS.PART_CELL_STATUS_COLOR, out2 => "DB8000_PART_STATUS".UNIT_03.FIXTURE_1.PART_A.STATUS.PART_MAIN_STATUS_COLOR)
   END_RUNG
   RUNG wire#w1
      Contact( "DB8000_PART_STATUS".UNIT_03.FIXTURE_1.PART_A.STATUS.PRESENT )
      wire#w2
      I_Contact( "DB8000_PART_STATUS".UNIT_03.FIXTURE_1.PART_A.STATUS.PART_REJECTED )
      I_Contact( "DB8000_PART_STATUS".UNIT_03.FIXTURE_1.PART_A.STATUS.QUALITY_PART )
      { S7_GenerateENO := "TRUE" } Move(in := 1, out1 => "DB8000_PART_STATUS".UNIT_03.FIXTURE_1.PART_A.STATUS.PART_MAIN_STATUS_COLOR, out2 => "DB2401_DBB_DEFINE".PART_STATUS.DBB_1096)
   END_RUNG
   RUNG wire#w2
      Contact( "DB8000_PART_STATUS".UNIT_03.FIXTURE_1.PART_A.STATUS.PART_REJECTED )
      { S7_GenerateENO := "TRUE" } Move(in := 2, out1 => "DB8000_PART_STATUS".UNIT_03.FIXTURE_1.PART_A.STATUS.PART_MAIN_STATUS_COLOR, out2 => "DB2401_DBB_DEFINE".PART_STATUS.DBB_1096)
   END_RUNG
   RUNG wire#w2
      Contact( "DB8000_PART_STATUS".UNIT_03.FIXTURE_1.PART_A.STATUS.QUALITY_PART )
      I_Contact( "DB8000_PART_STATUS".UNIT_03.FIXTURE_1.PART_A.STATUS.PART_REJECTED )
      { S7_GenerateENO := "TRUE" } Move(in := 3, out1 => "DB8000_PART_STATUS".UNIT_03.FIXTURE_1.PART_A.STATUS.PART_MAIN_STATUS_COLOR, out2 => "DB2401_DBB_DEFINE".PART_STATUS.DBB_1096)
   END_RUNG
   RUNG wire#w1
      Contact( "DB8000_PART_STATUS".UNIT_03.FIXTURE_1.PART_A.STATUS.PRESENT )
      wire#w3
      Contact( "DB8000_PART_STATUS".UNIT_03.FIXTURE_1.PART_A.STATUS.CELL_STATUS.NEW )
      { S7_GenerateENO := "TRUE" } Move(in := 1, out1 => "DB8000_PART_STATUS".UNIT_03.FIXTURE_1.PART_A.STATUS.PART_CELL_STATUS_COLOR, out2 => "DB2401_DBB_DEFINE".PART_STATUS.DBB_1096)
   END_RUNG
   RUNG wire#w3
      Contact( "DB8000_PART_STATUS".UNIT_03.FIXTURE_1.PART_A.STATUS.UNIT_01_STATUS.FACE_R_STATION_3_DONE )
      { S7_GenerateENO := "TRUE" } Move(in := 2, out1 => "DB8000_PART_STATUS".UNIT_03.FIXTURE_1.PART_A.STATUS.PART_CELL_STATUS_COLOR, out2 => "DB2401_DBB_DEFINE".PART_STATUS.DBB_1096)
   END_RUNG
   RUNG wire#w3
      Contact( "DB8000_PART_STATUS".UNIT_03.FIXTURE_1.PART_A.STATUS.UNIT_01_STATUS.FACE_R_STATION_4_DONE )
      { S7_GenerateENO := "TRUE" } Move(in := 3, out1 => "DB8000_PART_STATUS".UNIT_03.FIXTURE_1.PART_A.STATUS.PART_CELL_STATUS_COLOR, out2 => "DB2401_DBB_DEFINE".PART_STATUS.DBB_1096)
   END_RUNG
   RUNG wire#w3
      Contact( "DB8000_PART_STATUS".UNIT_03.FIXTURE_1.PART_A.STATUS.CELL_STATUS.U01_ONE_FACE_DONE_ROTATED )
      { S7_GenerateENO := "TRUE" } Move(in := 4, out1 => "DB8000_PART_STATUS".UNIT_03.FIXTURE_1.PART_A.STATUS.PART_CELL_STATUS_COLOR, out2 => "DB2401_DBB_DEFINE".PART_STATUS.DBB_1096)
   END_RUNG
   RUNG wire#w3
      Contact( "DB8000_PART_STATUS".UNIT_03.FIXTURE_1.PART_A.STATUS.UNIT_01_STATUS.FACE_N_STATION_3_DONE )
      { S7_GenerateENO := "TRUE" } Move(in := 5, out1 => "DB8000_PART_STATUS".UNIT_03.FIXTURE_1.PART_A.STATUS.PART_CELL_STATUS_COLOR, out2 => "DB2401_DBB_DEFINE".PART_STATUS.DBB_1096)
   END_RUNG
   RUNG wire#w3
      Contact( "DB8000_PART_STATUS".UNIT_03.FIXTURE_1.PART_A.STATUS.UNIT_01_STATUS.FACE_N_STATION_4_DONE )
      { S7_GenerateENO := "TRUE" } Move(in := 6, out1 => "DB8000_PART_STATUS".UNIT_03.FIXTURE_1.PART_A.STATUS.PART_CELL_STATUS_COLOR, out2 => "DB2401_DBB_DEFINE".PART_STATUS.DBB_1096)
   END_RUNG
   RUNG wire#w3
      Contact( "DB8000_PART_STATUS".UNIT_03.FIXTURE_1.PART_A.STATUS.CELL_STATUS.U01_DONE_IN_TRANSIT )
      { S7_GenerateENO := "TRUE" } Move(in := 7, out1 => "DB8000_PART_STATUS".UNIT_03.FIXTURE_1.PART_A.STATUS.PART_CELL_STATUS_COLOR, out2 => "DB2401_DBB_DEFINE".PART_STATUS.DBB_1096)
   END_RUNG
   RUNG wire#w3
      Contact( "DB8000_PART_STATUS".UNIT_03.FIXTURE_1.PART_A.STATUS.UNIT_02_STATUS.FACE_R_STATION_2_DONE )
      { S7_GenerateENO := "TRUE" } Move(in := 8, out1 => "DB8000_PART_STATUS".UNIT_03.FIXTURE_1.PART_A.STATUS.PART_CELL_STATUS_COLOR, out2 => "DB2401_DBB_DEFINE".PART_STATUS.DBB_1096)
   END_RUNG
   RUNG wire#w3
      Contact( "DB8000_PART_STATUS".UNIT_03.FIXTURE_1.PART_A.STATUS.UNIT_02_STATUS.FACE_R_STATION_3_DONE )
      Move(in := 9, out1 => "DB8000_PART_STATUS".UNIT_03.FIXTURE_1.PART_A.STATUS.PART_CELL_STATUS_COLOR, out2 => "DB2401_DBB_DEFINE".PART_STATUS.DBB_1096)
   END_RUNG
   RUNG wire#w3
      Contact( "DB8000_PART_STATUS".UNIT_03.FIXTURE_1.PART_A.STATUS.UNIT_02_STATUS.FACE_R_STATION_4_DONE )
      Move(in := 10, out1 => "DB8000_PART_STATUS".UNIT_03.FIXTURE_1.PART_A.STATUS.PART_CELL_STATUS_COLOR, out2 => "DB2401_DBB_DEFINE".PART_STATUS.DBB_1096)
   END_RUNG
   RUNG wire#w3
      Contact( "DB8000_PART_STATUS".UNIT_03.FIXTURE_1.PART_A.STATUS.CELL_STATUS.U02_ONE_FACE_DONE_ROTATED )
      Move(in := 11, out1 => "DB8000_PART_STATUS".UNIT_03.FIXTURE_1.PART_A.STATUS.PART_CELL_STATUS_COLOR, out2 => "DB2401_DBB_DEFINE".PART_STATUS.DBB_1096)
   END_RUNG
   RUNG wire#w3
      Contact( "DB8000_PART_STATUS".UNIT_03.FIXTURE_1.PART_A.STATUS.UNIT_02_STATUS.FACE_N_STATION_2_DONE )
      Move(in := 12, out1 => "DB8000_PART_STATUS".UNIT_03.FIXTURE_1.PART_A.STATUS.PART_CELL_STATUS_COLOR, out2 => "DB2401_DBB_DEFINE".PART_STATUS.DBB_1096)
   END_RUNG
   RUNG wire#w3
      Contact( "DB8000_PART_STATUS".UNIT_03.FIXTURE_1.PART_A.STATUS.UNIT_02_STATUS.FACE_N_STATION_3_DONE )
      Move(in := 13, out1 => "DB8000_PART_STATUS".UNIT_03.FIXTURE_1.PART_A.STATUS.PART_CELL_STATUS_COLOR, out2 => "DB2401_DBB_DEFINE".PART_STATUS.DBB_1096)
   END_RUNG
   RUNG wire#w3
      Contact( "DB8000_PART_STATUS".UNIT_03.FIXTURE_1.PART_A.STATUS.UNIT_02_STATUS.FACE_N_STATION_4_DONE )
      Move(in := 14, out1 => "DB8000_PART_STATUS".UNIT_03.FIXTURE_1.PART_A.STATUS.PART_CELL_STATUS_COLOR, out2 => "DB2401_DBB_DEFINE".PART_STATUS.DBB_1096)
   END_RUNG
   RUNG wire#w3
      Contact( "DB8000_PART_STATUS".UNIT_03.FIXTURE_1.PART_A.STATUS.CELL_STATUS.U02_DONE_IN_TRANSIT )
      Move(in := 15, out1 => "DB8000_PART_STATUS".UNIT_03.FIXTURE_1.PART_A.STATUS.PART_CELL_STATUS_COLOR, out2 => "DB2401_DBB_DEFINE".PART_STATUS.DBB_1096)
   END_RUNG
   RUNG wire#w3
      Contact( "DB8000_PART_STATUS".UNIT_03.FIXTURE_1.PART_A.STATUS.CELL_STATUS.COOLING_DONE )
      Move(in := 16, out1 => "DB8000_PART_STATUS".UNIT_03.FIXTURE_1.PART_A.STATUS.PART_CELL_STATUS_COLOR, out2 => "DB2401_DBB_DEFINE".PART_STATUS.DBB_1096)
   END_RUNG
   RUNG wire#w3
      Contact( "DB8000_PART_STATUS".UNIT_03.FIXTURE_1.PART_A.STATUS.CELL_STATUS.INSPECTION_DONE )
      Move(in := 17, out1 => "DB8000_PART_STATUS".UNIT_03.FIXTURE_1.PART_A.STATUS.PART_CELL_STATUS_COLOR, out2 => "DB2401_DBB_DEFINE".PART_STATUS.DBB_1096)
   END_RUNG
   // the same network as SCL:
   // ENO of a box is taken as its EN; it also drops when the box reports an error
   IF "M_ONE" AND NOT "DB8000_PART_STATUS".UNIT_03.FIXTURE_1.PART_A.STATUS.PRESENT THEN
       "DB2401_DBB_DEFINE".PART_STATUS.DBB_1096 := 0;
       "DB2401_DBB_DEFINE".PART_STATUS.DBB_1097 := 0;
       "DB8000_PART_STATUS".UNIT_03.FIXTURE_1.PART_A.STATUS.PART_CELL_STATUS_COLOR := 0;
       "DB8000_PART_STATUS".UNIT_03.FIXTURE_1.PART_A.STATUS.PART_MAIN_STATUS_COLOR := 0;
   END_IF;
   #_w1 := "M_ONE" AND "DB8000_PART_STATUS".UNIT_03.FIXTURE_1.PART_A.STATUS.PRESENT;
   IF #_w1 AND NOT "DB8000_PART_STATUS".UNIT_03.FIXTURE_1.PART_A.STATUS.PART_REJECTED AND NOT "DB8000_PART_STATUS".UNIT_03.FIXTURE_1.PART_A.STATUS.QUALITY_PART THEN
       "DB8000_PART_STATUS".UNIT_03.FIXTURE_1.PART_A.STATUS.PART_MAIN_STATUS_COLOR := 1;
       "DB2401_DBB_DEFINE".PART_STATUS.DBB_1096 := 1;
   END_IF;
   IF #_w1 AND "DB8000_PART_STATUS".UNIT_03.FIXTURE_1.PART_A.STATUS.PART_REJECTED THEN
       "DB8000_PART_STATUS".UNIT_03.FIXTURE_1.PART_A.STATUS.PART_MAIN_STATUS_COLOR := 2;
       "DB2401_DBB_DEFINE".PART_STATUS.DBB_1096 := 2;
   END_IF;
   IF #_w1 AND "DB8000_PART_STATUS".UNIT_03.FIXTURE_1.PART_A.STATUS.QUALITY_PART AND NOT "DB8000_PART_STATUS".UNIT_03.FIXTURE_1.PART_A.STATUS.PART_REJECTED THEN
       "DB8000_PART_STATUS".UNIT_03.FIXTURE_1.PART_A.STATUS.PART_MAIN_STATUS_COLOR := 3;
       "DB2401_DBB_DEFINE".PART_STATUS.DBB_1096 := 3;
   END_IF;
   #_w2 := "M_ONE" AND "DB8000_PART_STATUS".UNIT_03.FIXTURE_1.PART_A.STATUS.PRESENT;
   IF #_w2 AND "DB8000_PART_STATUS".UNIT_03.FIXTURE_1.PART_A.STATUS.CELL_STATUS.NEW THEN
       "DB8000_PART_STATUS".UNIT_03.FIXTURE_1.PART_A.STATUS.PART_CELL_STATUS_COLOR := 1;
       "DB2401_DBB_DEFINE".PART_STATUS.DBB_1096 := 1;
   END_IF;
   IF #_w2 AND "DB8000_PART_STATUS".UNIT_03.FIXTURE_1.PART_A.STATUS.UNIT_01_STATUS.FACE_R_STATION_3_DONE THEN
       "DB8000_PART_STATUS".UNIT_03.FIXTURE_1.PART_A.STATUS.PART_CELL_STATUS_COLOR := 2;
       "DB2401_DBB_DEFINE".PART_STATUS.DBB_1096 := 2;
   END_IF;
   IF #_w2 AND "DB8000_PART_STATUS".UNIT_03.FIXTURE_1.PART_A.STATUS.UNIT_01_STATUS.FACE_R_STATION_4_DONE THEN
       "DB8000_PART_STATUS".UNIT_03.FIXTURE_1.PART_A.STATUS.PART_CELL_STATUS_COLOR := 3;
       "DB2401_DBB_DEFINE".PART_STATUS.DBB_1096 := 3;
   END_IF;
   IF #_w2 AND "DB8000_PART_STATUS".UNIT_03.FIXTURE_1.PART_A.STATUS.CELL_STATUS.U01_ONE_FACE_DONE_ROTATED THEN
       "DB8000_PART_STATUS".UNIT_03.FIXTURE_1.PART_A.STATUS.PART_CELL_STATUS_COLOR := 4;
       "DB2401_DBB_DEFINE".PART_STATUS.DBB_1096 := 4;
   END_IF;
   IF #_w2 AND "DB8000_PART_STATUS".UNIT_03.FIXTURE_1.PART_A.STATUS.UNIT_01_STATUS.FACE_N_STATION_3_DONE THEN
       "DB8000_PART_STATUS".UNIT_03.FIXTURE_1.PART_A.STATUS.PART_CELL_STATUS_COLOR := 5;
       "DB2401_DBB_DEFINE".PART_STATUS.DBB_1096 := 5;
   END_IF;
   IF #_w2 AND "DB8000_PART_STATUS".UNIT_03.FIXTURE_1.PART_A.STATUS.UNIT_01_STATUS.FACE_N_STATION_4_DONE THEN
       "DB8000_PART_STATUS".UNIT_03.FIXTURE_1.PART_A.STATUS.PART_CELL_STATUS_COLOR := 6;
       "DB2401_DBB_DEFINE".PART_STATUS.DBB_1096 := 6;
   END_IF;
   IF #_w2 AND "DB8000_PART_STATUS".UNIT_03.FIXTURE_1.PART_A.STATUS.CELL_STATUS.U01_DONE_IN_TRANSIT THEN
       "DB8000_PART_STATUS".UNIT_03.FIXTURE_1.PART_A.STATUS.PART_CELL_STATUS_COLOR := 7;
       "DB2401_DBB_DEFINE".PART_STATUS.DBB_1096 := 7;
   END_IF;
   IF #_w2 AND "DB8000_PART_STATUS".UNIT_03.FIXTURE_1.PART_A.STATUS.UNIT_02_STATUS.FACE_R_STATION_2_DONE THEN
       "DB8000_PART_STATUS".UNIT_03.FIXTURE_1.PART_A.STATUS.PART_CELL_STATUS_COLOR := 8;
       "DB2401_DBB_DEFINE".PART_STATUS.DBB_1096 := 8;
   END_IF;
   IF #_w2 AND "DB8000_PART_STATUS".UNIT_03.FIXTURE_1.PART_A.STATUS.UNIT_02_STATUS.FACE_R_STATION_3_DONE THEN
       "DB8000_PART_STATUS".UNIT_03.FIXTURE_1.PART_A.STATUS.PART_CELL_STATUS_COLOR := 9;
       "DB2401_DBB_DEFINE".PART_STATUS.DBB_1096 := 9;
   END_IF;
   IF #_w2 AND "DB8000_PART_STATUS".UNIT_03.FIXTURE_1.PART_A.STATUS.UNIT_02_STATUS.FACE_R_STATION_4_DONE THEN
       "DB8000_PART_STATUS".UNIT_03.FIXTURE_1.PART_A.STATUS.PART_CELL_STATUS_COLOR := 10;
       "DB2401_DBB_DEFINE".PART_STATUS.DBB_1096 := 10;
   END_IF;
   IF #_w2 AND "DB8000_PART_STATUS".UNIT_03.FIXTURE_1.PART_A.STATUS.CELL_STATUS.U02_ONE_FACE_DONE_ROTATED THEN
       "DB8000_PART_STATUS".UNIT_03.FIXTURE_1.PART_A.STATUS.PART_CELL_STATUS_COLOR := 11;
       "DB2401_DBB_DEFINE".PART_STATUS.DBB_1096 := 11;
   END_IF;
   IF #_w2 AND "DB8000_PART_STATUS".UNIT_03.FIXTURE_1.PART_A.STATUS.UNIT_02_STATUS.FACE_N_STATION_2_DONE THEN
       "DB8000_PART_STATUS".UNIT_03.FIXTURE_1.PART_A.STATUS.PART_CELL_STATUS_COLOR := 12;
       "DB2401_DBB_DEFINE".PART_STATUS.DBB_1096 := 12;
   END_IF;
   IF #_w2 AND "DB8000_PART_STATUS".UNIT_03.FIXTURE_1.PART_A.STATUS.UNIT_02_STATUS.FACE_N_STATION_3_DONE THEN
       "DB8000_PART_STATUS".UNIT_03.FIXTURE_1.PART_A.STATUS.PART_CELL_STATUS_COLOR := 13;
       "DB2401_DBB_DEFINE".PART_STATUS.DBB_1096 := 13;
   END_IF;
   IF #_w2 AND "DB8000_PART_STATUS".UNIT_03.FIXTURE_1.PART_A.STATUS.UNIT_02_STATUS.FACE_N_STATION_4_DONE THEN
       "DB8000_PART_STATUS".UNIT_03.FIXTURE_1.PART_A.STATUS.PART_CELL_STATUS_COLOR := 14;
       "DB2401_DBB_DEFINE".PART_STATUS.DBB_1096 := 14;
   END_IF;
   IF #_w2 AND "DB8000_PART_STATUS".UNIT_03.FIXTURE_1.PART_A.STATUS.CELL_STATUS.U02_DONE_IN_TRANSIT THEN
       "DB8000_PART_STATUS".UNIT_03.FIXTURE_1.PART_A.STATUS.PART_CELL_STATUS_COLOR := 15;
       "DB2401_DBB_DEFINE".PART_STATUS.DBB_1096 := 15;
   END_IF;
   IF #_w2 AND "DB8000_PART_STATUS".UNIT_03.FIXTURE_1.PART_A.STATUS.CELL_STATUS.COOLING_DONE THEN
       "DB8000_PART_STATUS".UNIT_03.FIXTURE_1.PART_A.STATUS.PART_CELL_STATUS_COLOR := 16;
       "DB2401_DBB_DEFINE".PART_STATUS.DBB_1096 := 16;
   END_IF;
   IF #_w2 AND "DB8000_PART_STATUS".UNIT_03.FIXTURE_1.PART_A.STATUS.CELL_STATUS.INSPECTION_DONE THEN
       "DB8000_PART_STATUS".UNIT_03.FIXTURE_1.PART_A.STATUS.PART_CELL_STATUS_COLOR := 17;
       "DB2401_DBB_DEFINE".PART_STATUS.DBB_1096 := 17;
   END_IF;
END_REGION
END_FUNCTION
